// TwinCAT 3 PLC project plc_greenmirror
// ProgramVersion: 3.1.4024.0
// libraries:
//   Tc2_Standard, * (Beckhoff Automation GmbH)
//   Tc2_System, * (Beckhoff Automation GmbH)
//   Tc3_Module, * (Beckhoff Automation GmbH)
//   VisuSymbols,3.5.10.0,System
// project tree:
//   / GlobalTextList.TcGTLO, lightControl_1.TcTTO, PlcTask.TcTTO, timerControl_1.TcTTO, Visualization Manager.TcVMO (not stored)
//   GVLs/ GVL.TcGVL
//   POUs/ checkDistance.TcPOU, lightControl.TcPOU, MAIN.TcPOU, timerControl.TcPOU
//   VISUs/ Visualization.TcVIS
// real-time tasks:
//   TASK PlcTask: cycle T#10ms, priority 20, ADS port 350
//   TASK lightControl: cycle T#10ms, priority 21, ADS port 351
//   TASK timerControl: cycle T#10ms, priority 22, ADS port 352

CONFIGURATION plc_greenmirror
    RESOURCE PLC ON TwinCAT3
        TASK lightControl_1(INTERVAL := T#10ms, PRIORITY := 21);
        TASK PlcTask(INTERVAL := T#10ms, PRIORITY := 20);
        TASK timerControl_1(INTERVAL := T#10ms, PRIORITY := 22);
        PROGRAM lightControl WITH lightControl_1 : lightControl;
        PROGRAM MAIN WITH PlcTask : MAIN;
        PROGRAM timerControl WITH timerControl_1 : timerControl;
    END_RESOURCE
END_CONFIGURATION

// ---- GVLs/GVL.TcGVL
{attribute 'qualified_only'}
VAR_GLOBAL
	distance : REAL := 0.0;        // Distance between user and mirror in meters
    lightStatus : BOOL := FALSE;   // Light status (ON/OFF)
    timerActive : BOOL := FALSE;   // Timer active status
    timerElapsed : BOOL := FALSE;  // Timer finished status
END_VAR

// ---- POUs/lightControl.TcPOU
PROGRAM lightControl
VAR
    userNearMirror : BOOL;  // Variable to store whether the user is near the mirror
END_VAR

// Call the function to check if the user is near the mirror
userNearMirror := checkDistance(distance_in_function := GVL.distance);

// Turn on the light if the user is near the mirror
IF userNearMirror = TRUE THEN
    GVL.lightStatus := TRUE;
ELSIF userNearMirror = FALSE THEN
    // Start the timer when the user moves away from the mirror
    timerControl();  
END_IF

END_PROGRAM

// ---- POUs/checkDistance.TcPOU
FUNCTION checkDistance : BOOL
VAR_INPUT
    distance_in_function : REAL;  // Distance from the mirror
END_VAR

// If the distance is less than or equal to 1 meter, return TRUE, else return FALSE
IF distance_in_function<= 1.0 THEN
    checkDistance := TRUE;
ELSE
    checkDistance := FALSE;
END_IF

END_FUNCTION

// ---- POUs/timerControl.TcPOU
PROGRAM timerControl
VAR
	 timer : TOF;  // Timer off-delay function block
END_VAR

// Start the TOF timer if the user moves away (light is still on) and the timer hasn't started
IF GVL.lightStatus = TRUE AND GVL.timerActive = FALSE THEN
    GVL.timerActive := TRUE;
    timer(IN := TRUE, PT := T#15s);  // Start 15-second off-delay timer
END_IF

// If the timer finishes (Q goes TRUE), turn off the light
IF timer.Q THEN
    GVL.lightStatus := FALSE;  // Turn off the light after 15s delay
    GVL.timerActive := FALSE;  // Reset the timer state
END_IF

// Reset the timer when the light is off (if the user moves away before timer completes)
IF GVL.lightStatus = FALSE THEN
    timer(IN := FALSE);  // Stop the timer
    GVL.timerActive := FALSE;  // Reset timer active status
END_IF

END_PROGRAM

// ---- POUs/MAIN.TcPOU
PROGRAM MAIN
VAR
END_VAR

lightControl();
timerControl();

END_PROGRAM

// ---- VISUs/Visualization.TcVIS
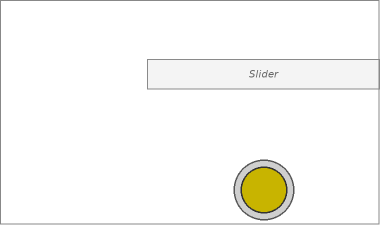
VISUALIZATION Visualization  // 380x225
    Lamp1 (229,155 70x70), variable: GVL.lightStatus, style: Lamp-Lamp1-Yellow
    Slider (147,59 233x30), variable: GVL.distance, scale 0..5
END_VISUALIZATION
